PROGRAM Main
VAR
 	fbPowerMaster : FB_PowerMaster;
  fbPowerAxis1 : FB_PowerAxis1;
  
  fbTestAxle : FB_testAxle;
  
  //Axis day 2 training
  myAxisA : FB_Axis;
	myAxisB : FB_Axis;
	myAxisVirtual : FB_Axis;
	myAxisStepper : FB_Axis;
	fbAxisStMachine : FB_AxisStMachine;
END_VAR

//Axis day 2 training
//myAxisA(AxisInOut := GVL.Axis_servoA);
//myAxisB(AxisInOut := GVL.Axis_servoB);
//myAxisVirtual(AxisInOut := GVL.Axis_servoVirtual);
//myAxisStepper(AxisInOut := GVL.Axis_servo);
//fbAxisStMachine(AxisInOut := GVL.Axis_servoA);

//fbPowerAxis1();
fbPowerMaster();

//fbTestAxle();

END_PROGRAM

(* stored: Version 1.1.0.1, ProductVersion 3.1.4024.12
   POU Main: Id {b2f2a346-2aab-4873-ae80-3f4daff09e02}, SpecialFunc None *)
